FUNCTION_BLOCK FB_AT1K2_PositionState EXTENDS FB_PositionStateInOut

VAR
    bInitialized: BOOL := FALSE;
END_VAR

IF NOT bInitialized THEN
    bInitialized := TRUE;

    arrStates[1] := stOut;
    arrStates[2] := stIn;
	
END_IF
setState := enumSet;
Exec();
enumGet := getState;
enumSet := setState;

END_FUNCTION_BLOCK

(* stored: Version 1.1.0.1, ProductVersion 3.1.4022.18
   POU FB_AT1K2_PositionState: Id {7d06e279-8ae9-4efc-8581-65b6fed1a960}, SpecialFunc None *)
